Staubli VAL3: RobotPolish.dtx

bool bBIO[32]
  [16] = true
  [18] = true
  [22] = true
bool bDebug_PC[6] = true
bool bExit
bool bForceError
bool bHome
bool bInterVal
bool bIsAlarm
bool bIsPower
bool bJntOrPtSpd
bool bOverRun
bool bPause
bool bRefreshMsg[6]
  [0] = true
  [1] = true
  [2] = true
  [3] = true
  [4] = true
  [5] = true
bool bSuspend
bool bTableAlm
bool bTxtLoad
bool bUpload
bool bZero
frame fFrame = {x=1612.970915, y=39.891118, z=-82.912831, rx=0.071185, ry=-0.543234, rz=-77.228709, fatherId=world[0]}
jointRx jCurrentJoint
jointRx jHome = {j1=40.634813, j2=24.616005, j3=104.715218, j4=-108.663007, j5=68.526435, j6=132.709111}
jointRx jJHome = {j1=40.634813, j2=24.616005, j3=104.715218, j4=-108.663007, j5=68.526435, j6=132.709111}
mdesc mNomSpeed = {accel=36, vel=60, decel=36, rmax=2000, tmax=100, blend=cartesian, leave=5, reach=5}
num nATIPress
num nATiPressBuff
num nFunctionIndex = -1
num nInterfaceType = 9
num nJntList = 5
public num nLimitAti[6]
  [0] = 500
  [1] = 500
  [2] = 500
  [3] = 100
  [4] = 100
  [5] = 100
num nMoveID
num nPage
num nPauseTime = 6
num nSelect
num nTabSpeed = 5
num nTimeBuff = 6728.108
num nTxtSelseted = 1
num nVirtualKey = -1
num nWorkModeStatus = 2
num nWorkingMode = 4
pointRx p = {x=-96.25, y=181, rx=-8.631, ry=175.438, rz=-89.108, fatherId=fFrame[0]}
pointRx pCurrent = {x=-182.218267, y=-975.12613, z=2269.00101, rx=89.444006, ry=167.500069, rz=-89.947529, shoulder=lefty, elbow=epositive, wrist=wpositive, fatherId=fFrame[0]}
string sButtons[2]
  [0] = "Yes"
  [1] = "No"
string sErrorMsg[8]
  [0] = "UPS报错，检查工厂供电"
  [1] = "转台故障报警"
  [2] = "工具报警"
  [3] = "ATI与机器人通讯异常"
  [4] = "打磨力超出上限"
  [5] = "急停状态激活中"
string sItems[8]
  [0] = "信号"
  [1] = "生产"
  [2] = "TCP"
  [3] = "Frame"
  [4] = "Home"
  [5] = "速度"
  [7] = "退出"
string sMassage
string sPrdStatus[10]
  [0] = "Txt文件:"
  [1] = "OAP275_Test.txt"
  [2] = "生产状态:无生产"
  [3] = "运动状态:Move"
  [4] = "总路径个数:     1"
  [5] = "当前路径  :     1"
  [6] = "写入点个数:     9"
  [7] = "读取点个数:     9"
  [8] = "当前MoveID:     9"
  [9] = "瞬时速度  :  0   "
string sStrFileName[5]
string sTxtLists[12]
  [0] = "Test.txt"
  [1] = "Test2.txt"
string sTxtSelected = "OAP275_Test.txt"
tool tTTool = {x=-12.113679, y=2.514779, z=192.872851, rx=33.798326, ry=31.269905, rz=-56.042932, fatherId=flange[0], ioLink=valve1}
public tool tTool = {x=350.22, y=-0.767094, z=232.538993, rx=-89.841339, ry=89.729222, rz=89.842087, fatherId=flange[0], ioLink=valve1}
trsf trFrame = {x=1612.647528, y=43.391654, z=-98.162922, rx=0.062117, ry=-0.932889, rz=-75.762654}
